PROGRAM MAIN
VAR
	bRunning : BOOL;
END_VAR

END_PROGRAM

(* stored: Version 1.1.0.1, ProductVersion 3.1.4024.16
   POU MAIN: Id {d44c1382-4994-441d-a73c-18d086b6e431}, SpecialFunc None *)
